PROGRAM HMISimulation
VAR
	
fbHMIJoystick : FB_HMISimulationJoystick;
fbNotEnabled : FB_NotEnabled;
fbEnabled : FB_Enabled;
fbVelFeedForward : FB_OpenLoopControl;
END_VAR


IF HMIinput.bHMIPowerSwitch = FALSE THEN //When power is off
		
	fbNotEnabled();
	
ELSIF HMIinput.bHMIPowerSwitch = TRUE THEN // When power is on

	fbEnabled();

END_IF

// In real system, the modes is their own boolean value. "Rotary Switch" on HMI
IF HMIInput.bHMIModeSwitch = FALSE AND HMIInput.bHMIStartSwitch = TRUE AND HMIInput.bHMIStopSwitch = FALSE THEN
	
	fbHMIJoystick();
	fbVelFeedForward ();

END_IF

END_PROGRAM

(* stored: Version 1.1.0.1, ProductVersion 3.1.4024.10
   POU HMISimulation: Id {66b8bd2b-e4eb-40d8-ae53-cdc86fa23b3a}, SpecialFunc None *)
